INTERFACE ITF_PMLModuleBase

PROPERTY ActualProductionRate : LREAL
GET
END_GET
END_PROPERTY

PROPERTY AncestorIDs : STRING
GET
END_GET
SET
END_SET
END_PROPERTY

METHOD CyclicLogic
END_METHOD

PROPERTY Enabled : BOOL
GET
END_GET
SET
END_SET
END_PROPERTY

PROPERTY LogModeChanges : BOOL
GET
END_GET
SET
END_SET
END_PROPERTY

PROPERTY LogStateChanges : BOOL
GET
END_GET
SET
END_SET
END_PROPERTY

PROPERTY MasterDataStructure_Adder :  ITF_Tree_IndexBased
GET
END_GET
SET
END_SET
END_PROPERTY

PROPERTY Mode : E_PMLUnitMode
GET
END_GET
END_PROPERTY

PROPERTY ModeCommand : DINT
SET
END_SET
END_PROPERTY

PROPERTY ModuleID : UDINT
GET
END_GET
SET
END_SET
END_PROPERTY

PROPERTY ModuleName : STRING
GET
END_GET
SET
END_SET
END_PROPERTY

PROPERTY SimulateAllChildren : BOOL
GET
END_GET
SET
END_SET
END_PROPERTY

PROPERTY State : E_PMLState
GET
END_GET
END_PROPERTY

PROPERTY StateCommand : E_PMLCommand
SET
END_SET
END_PROPERTY

PROPERTY TargetProductionRate : LREAL
GET
END_GET
SET
END_SET
END_PROPERTY

END_INTERFACE

(* stored: Version 1.1.0.1, ProductVersion 3.1.4024.9
   Itf ITF_PMLModuleBase: Id {eca4a56b-850e-483e-b687-2de3b3950c24}
   Folder 01_Properties: Id {b9b76dff-8c1e-4a81-8fb8-90bae0384924}
   Folder 01_Config: Id {c034098c-56e3-4732-a681-b27df2a6a3ee}
   Folder 02_Control: Id {f156f415-4f70-402d-872f-de20fbc04916}
   Folder 03_Status: Id {681bf848-54e8-410c-a596-7e58d3fea268}
   Folder 02_Methods: Id {fbb15efd-8a92-4fbb-a79e-6108b9c86638}
   Property ActualProductionRate: Id {7ed2842f-7cd7-4694-89fa-c274118f161d}
   Get Get: Id {d58d319d-6658-4d0d-a426-5afa6e67b86d}
   Property AncestorIDs: Id {ddc4ec9f-03b5-4a9a-9708-c7ae158f5b04}
   Get Get: Id {f334f915-3beb-484a-b889-7d0a10f7ff80}
   Set Set: Id {6f7535d2-f023-4f68-b8d5-8ced32bad9bc}
   Method CyclicLogic: Id {93d2f113-3cbc-4b7f-a56f-610da986a3d8}
   Property Enabled: Id {d2ef8559-89f7-4b1a-8a7a-48174a953874}
   Get Get: Id {54ba9b0b-2822-4ef3-b25b-9c30c5987360}
   Set Set: Id {c6163e65-6cf3-4a30-a648-3de95a4476c4}
   Property LogModeChanges: Id {3ebf3a99-dead-418c-b471-054c7c8d6544}
   Get Get: Id {e04dfd29-bd9f-4f54-828e-2fc4045c23bc}
   Set Set: Id {1785a2f9-a528-437d-84c4-405797055f1f}
   Property LogStateChanges: Id {1b008608-b316-4d3a-ba87-f437076859ca}
   Get Get: Id {66bc6c53-f9e2-4511-89b6-29fb383f77e7}
   Set Set: Id {a9b78c0c-4b3e-4169-a6c7-77bf1bd91d29}
   Property MasterDataStructure_Adder: Id {e8e1f737-2d53-4f7e-85f8-3eda713a980e}
   Get Get: Id {9a79581e-ec99-41c5-b4c5-b12242225d5c}
   Set Set: Id {64ba5fdd-6f11-47c3-b21d-50cd6159df0d}
   Property Mode: Id {68aa19f0-a027-4849-bb10-f5584ab8d043}
   Get Get: Id {e4c0be11-49fb-4f99-95fb-f87a759ebdeb}
   Property ModeCommand: Id {11907bf7-f645-420b-85af-3bf0127cd7f1}
   Set Set: Id {0cf2eb2e-aedc-4e54-afcc-be209278627f}
   Property ModuleID: Id {b15ae476-29f6-49b3-bc0b-8d8de1f9a2ad}
   Get Get: Id {15915578-ed14-421a-b902-68fca348c24a}
   Set Set: Id {2e8dc440-ac63-48e1-b6bf-7bd9cd9ed340}
   Property ModuleName: Id {da8f2502-5e83-49c9-bcb7-07c02f3fcb7b}
   Get Get: Id {c93e64d6-b7f5-4fa1-96b7-7e8cdadc8f67}
   Set Set: Id {0e6ed32b-5954-42fd-b96a-59359710d227}
   Property SimulateAllChildren: Id {372d62d1-e10f-492d-bcb6-f6da619c14bf}
   Get Get: Id {84230418-3f62-4b95-99de-b381b48139b5}
   Set Set: Id {c531c7fa-5d73-4c05-905b-cee2a27a5492}
   Property State: Id {43595dac-7213-416e-a39c-be01c96ab13c}
   Get Get: Id {21f6fac7-5f70-4bd9-8ec4-66822702fbf5}
   Property StateCommand: Id {1c454ada-e18d-4933-8772-ef90079bfec6}
   Set Set: Id {3495e55a-b4ad-4161-a7ba-1793fe13d390}
   Property TargetProductionRate: Id {40ff0130-155a-47ee-8753-64a2da899a2d}
   Get Get: Id {7999c80a-1e65-4223-a767-fe3d703ca7f7}
   Set Set: Id {e468dc00-076e-4592-bf4e-e79c036a39bf} *)
